// TIA Portal V18 export
TYPE "PartData_UDT"
// stored: IsFailsafeCompliant false
   STRUCT
      PartDataHMI { S7_SetPoint := 'True'} : "PartDataHMI";   // 显示料盒编号
      PartBoxDataRecive : "PartCodeStruct_UDT";   // 扫码接收的物料信息
      PartBoxData { S7_SetPoint := 'True'} : Array[0..10] of "PartCodeStruct_UDT";   // 缓存的物料信息
      PartBoxDataNull : "PartCodeStruct_UDT";   // 空的物料信息
   END_STRUCT;
   // // PartBoxData[0] : 当前使用的物料信息
   // // PartBoxData[1] : 缓存1的物料信息
   // // PartBoxData[2] : 缓存2的物料信息
   // // PartBoxData[3] : 缓存3的物料信息
   // // PartBoxData[4] : 缓存4的物料信息
   // // PartBoxData[5] : 缓存5的物料信息
   // // PartBoxData[6] : 缓存6的物料信息
   // // PartBoxData[7] : 缓存7的物料信息
END_TYPE
